{attribute 'GeneratedUsingTerminal: EK1100-0000-0018'}
{attribute addProperty BoxType "EK1100-0000-0018"}
{attribute addProperty Id "Beckhoff_EL2xxxEK1122Beckhoff_EL2xxxEK1122_964E41392A_0001_EL2002_0000_0000EL2002_B02149405A_0002_EL2002_0000_0016EL2002_B02149405A_0003_EL2002_0000_0017EL2002_B02149405A_0004_EL2002_0000_0018EL2002_B02149405A_0005_EL2004_0000_0000EL2004_7B64371E7A_0006_EL2004_0000_0016EL2004_7B64371E7A_0007_EL2004_0000_0017EL2004_7B64371E7A_0008_EL2004_0000_0018EL2004_7B64371E7A_0009_EL2008_0000_0016EL2008_E2806B9511A_0010_EL2008_0000_0017EL2008_E2806B9511A_0011_EL2008_0000_0018EL2008_E2806B9511A_0012_EL2014_0000_0016EL2014_12F3E4E336A_0013_EL2014_0000_0017EL2014_12F3E4E336A_0014_EL2022_0000_0016EL2022_B02149405A_0015_EL2022_0000_0017EL2022_B02149405A_0016_EL2022_0000_0018EL2022_B02149405A_0017_EL2024_0000_0016EL2024_7B64371E7A_0018_EL2024_0000_0017EL2024_7B64371E7A_0019_EL2024_0000_0018EL2024_7B64371E7A_0020_EL2024_0000_0019EL2024_7B64371E7A_0021_EL2024_0010_0016EL2024_7B64371E7A_0022_EL2024_0010_0017EL2024_7B64371E7A_0023_EL2024_0010_0018EL2024_7B64371E7A_0024_EL2032_0000_0000EL2032_4C3AB2A48A_0025_EL2032_0000_0016EL2032_4C3AB2A48A_0026_EL2032_0000_0017EL2032_4C3AB2A48A_0027_EL2032_0000_0018EL2032_4C3AB2A48A_0028_EL2034_0000_0016EL2034_9227BD0712A_0029_EL2034_0000_0017EL2034_9227BD0712A_0030_EL2034_0000_0018EL2034_9227BD0712A_0031_EL2042_0000_0016EL2042_B02149405A_0032_EL2042_0000_0017EL2042_B02149405A_0033_EL2042_0000_0018EL2042_B02149405A_0034_EL2044_0000_0016EL2044_12F3E4E336A_0035_EL2084_0000_0016EL2084_7B64371E7A_0036_EL2084_0000_0017EL2084_7B64371E7A_0037_EL2084_0000_0018EL2084_7B64371E7A_0038_EL2088_0000_0016EL2088_E2806B9511A_0039_EL2088_0000_0017EL2088_E2806B9511A_0040_EL2088_0000_0018EL2088_E2806B9511A_0041_EL2124_0000_0016EL2124_7B64371E7A_0042_EL2124_0000_0017EL2124_7B64371E7A_0043_EL2124_0000_0018EL2124_7B64371E7A_0044_EL2202_0000_0000EL2202_B02149405A_0045_EL2202_0000_0016EL2202_E4D0F2567A_0046_EL2202_0000_0017EL2202_E4D0F2567A_0047_EL2202_0000_0018EL2202_E4D0F2567A_0048_EL2202_0000_0019EL2202_E4D0F2567A_0049_EL2202_0100_0016EL2202_FB12F0C615A_0050_EL2202_0100_0017EL2202_FB12F0C615A_0051_EL2202_0100_0018EL2202_FB12F0C615A_0052_EL2202_0100_0019EL2202_FB12F0C615A_0053_EL2212_0000_0018EL2212_25BC0E0A32A_0054_EL2212_0000_0019EL2212_25BC0E0A32A_0055_EL2212_0000_0020EL2212_C6DE676634A_0056_EL2212_0000_0021EL2212_C6DE676634A_0057_EL2212_0000_0022EL2212_C6DE676634A_0058_EL2212_0000_0023EL2212_C6DE676634A_0059_EL2252_0000_0000EL2252_FF939DB018A_0060_EL2252_0000_0016EL2252_BD1134C622A_0061_EL2252_0000_0017EL2252_F49A8E9224A_0062_EL2252_0000_0018EL2252_F49A8E9224A_0063_EL2252_0000_0019EL2252_F49A8E9224A_0064_EL2252_0000_0020EL2252_F49A8E9224A_0065_EL2258_0000_0016EL2258_1A7A2033508A_0066_EL2258_0000_0017EL2258_41B36B91516A_0067_EL2262_0000_0000EL2262_4683CFC914A_0068_EL2262_0000_0001EL2262_79C970B117A_0069_EL2262_0000_0002EL2262_147DB6E135A_0070_EL2262_0000_0003EL2262_147DB6E135A_0071_EL2262_0000_0004EL2262_9619875D40A_0072_EL2602_0000_0016EL2602_B02149405A_0073_EL2602_0000_0017EL2602_B02149405A_0074_EL2602_0000_0018EL2602_B02149405A_0075_EL2602_0010_0016EL2602_47E63F277A_0076_EL2612_0000_0016EL2612_B02149405A_0077_EL2612_0000_0017EL2612_B02149405A_0078_EL2612_0000_0018EL2612_B02149405A_0079_EL2622_0000_0016EL2622_B02149405A_0080_EL2622_0000_0017EL2622_B02149405A_0081_EL2622_0000_0018EL2622_B02149405A_0082_EL2622_0010_0016EL2622_47E63F277A_0083_EL2624_0000_0016EL2624_7B64371E7A_0084_EL2624_0000_0017EL2624_7B64371E7A_0085_EL2624_0000_0018EL2624_7B64371E7A_0086_EL2634_0000_0016EL2634_7B64371E7A_0087_EL2634_0000_0017EL2634_7B64371E7A_0088_EL2642_0000_0016EL2642_C5F9ACE731A_0089_EL2652_0000_0016EL2652_B02149405A_0090_EL2652_0000_0017EL2652_B02149405A_0091_EL2652_0000_0018EL2652_B02149405A_0092_EL2712_0000_0016EL2712_B02149405A_0093_EL2712_0000_0017EL2712_B02149405A_0094_EL2722_0000_0016EL2722_B02149405A_0095_EL2722_0010_0016EL2722_B02149405A_0096_EL2732_0000_0016EL2732_B02149405A_0097_EL2784_0000_0016EL2784_7B64371E7A_0098_EL2788_0000_0016EL2788_E2806B9511A_0099_EL2794_0000_0016EL2794_7B64371E7A_0100_EL2798_0000_0016EL2798_E2806B9511A_0101_EL2798_0000_0017EL2798_E2806B9511A_0102_EL2798_0000_0018EL2798_E2806B9511A_0103_EL2808_0000_0016EL2808_E2806B9511A_0104_EL2808_0000_0017EL2808_E2806B9511A_0105_EL2808_0000_0018EL2808_E2806B9511A_0106_EL2809_0000_0016EL2809_2B6483BD19A_0107_EL2809_0000_0017EL2809_2B6483BD19A_0108_EL2809_0000_0018EL2809_2B6483BD19A_0109_EL2819_0000_0016EL2819_3C4AB9A796A_0110_EL2819_0000_0017EL2819_3C4AB9A796A_0111_EL2819_0000_0018EL2819_3C4AB9A796A_0112_EL2828_0000_0016EL2828_E2806B9511A_0113_EL2828_0000_0017EL2828_E2806B9511A_0114_EL2872_0000_0016EL2872_2B6483BD19A_0115_EL2872_0000_0017EL2872_2B6483BD19A_0116_EL2872_0000_0018EL2872_2B6483BD19A_0117_EL2872_0000_0019EL2872_2B6483BD19A_0118_EL2872_0010_0016EL2872_2B6483BD19A_0119_EL2872_0010_0017EL2872_2B6483BD19A_0120_EL2872_0010_0018EL2872_2B6483BD19A_0121_EL2872_0010_0019EL2872_2B6483BD19A_0122_EL2878_0005_0016EL2878_76DE585D13A_0123_EL2889_0000_0016EL2889_2B6483BD19A_0124_EL2889_0000_0017EL2889_2B6483BD19A_0125_EL2889_0000_0018EL2889_2B6483BD19A_0126_ELM2642_0000_0016ELM2642_AD2D58FD31A_0127_ELM2644_0000_0016ELM2644_9E566A2A39A_0128_ELM2742_0000_0016ELM2742_AD2D58FD31A_0129_ELM2744_0000_0016ELM2744_9E566A2A39"}
{attribute addProperty CRC "4106566090"}
{attribute addProperty Size "2992"}
TYPE Beckhoff_EL2xxx_F4C539CA EXTENDS EK1100_1FC0878B :
STRUCT
	{attribute addProperty Name "Beckhoff EL2xxxEK1122"}
	{attribute addProperty PreviousPort "Beckhoff EL2xxx : B"}
	Beckhoff_EL2xxxEK1122 : Beckhoff_EL2xxxEK1122_964E4139;
	{attribute addProperty Name "A_0001(EL2002-0000-0000)"}
	{attribute addProperty PreviousPort "Beckhoff EL2xxxEK1122 : C"}
	A_0001_EL2002_0000_0000 : EL2002_B0214940;
	{attribute addProperty Name "A_0002(EL2002-0000-0016)"}
	{attribute addProperty PreviousPort "A_0001(EL2002-0000-0000) : B"}
	A_0002_EL2002_0000_0016 : EL2002_B0214940;
	{attribute addProperty Name "A_0003(EL2002-0000-0017)"}
	{attribute addProperty PreviousPort "A_0002(EL2002-0000-0016) : B"}
	A_0003_EL2002_0000_0017 : EL2002_B0214940;
	{attribute addProperty Name "A_0004(EL2002-0000-0018)"}
	{attribute addProperty PreviousPort "A_0003(EL2002-0000-0017) : B"}
	A_0004_EL2002_0000_0018 : EL2002_B0214940;
	{attribute addProperty Name "A_0005(EL2004-0000-0000)"}
	{attribute addProperty PreviousPort "A_0004(EL2002-0000-0018) : B"}
	A_0005_EL2004_0000_0000 : EL2004_7B64371E;
	{attribute addProperty Name "A_0006(EL2004-0000-0016)"}
	{attribute addProperty PreviousPort "A_0005(EL2004-0000-0000) : B"}
	A_0006_EL2004_0000_0016 : EL2004_7B64371E;
	{attribute addProperty Name "A_0007(EL2004-0000-0017)"}
	{attribute addProperty PreviousPort "A_0006(EL2004-0000-0016) : B"}
	A_0007_EL2004_0000_0017 : EL2004_7B64371E;
	{attribute addProperty Name "A_0008(EL2004-0000-0018)"}
	{attribute addProperty PreviousPort "A_0007(EL2004-0000-0017) : B"}
	A_0008_EL2004_0000_0018 : EL2004_7B64371E;
	{attribute addProperty Name "A_0009(EL2008-0000-0016)"}
	{attribute addProperty PreviousPort "A_0008(EL2004-0000-0018) : B"}
	A_0009_EL2008_0000_0016 : EL2008_E2806B95;
	{attribute addProperty Name "A_0010(EL2008-0000-0017)"}
	{attribute addProperty PreviousPort "A_0009(EL2008-0000-0016) : B"}
	A_0010_EL2008_0000_0017 : EL2008_E2806B95;
	{attribute addProperty Name "A_0011(EL2008-0000-0018)"}
	{attribute addProperty PreviousPort "A_0010(EL2008-0000-0017) : B"}
	A_0011_EL2008_0000_0018 : EL2008_E2806B95;
	{attribute addProperty Name "A_0012(EL2014-0000-0016)"}
	{attribute addProperty PreviousPort "A_0011(EL2008-0000-0018) : B"}
	A_0012_EL2014_0000_0016 : EL2014_12F3E4E3;
	{attribute addProperty Name "A_0013(EL2014-0000-0017)"}
	{attribute addProperty PreviousPort "A_0012(EL2014-0000-0016) : B"}
	A_0013_EL2014_0000_0017 : EL2014_12F3E4E3;
	{attribute addProperty Name "A_0014(EL2022-0000-0016)"}
	{attribute addProperty PreviousPort "A_0013(EL2014-0000-0017) : B"}
	A_0014_EL2022_0000_0016 : EL2022_B0214940;
	{attribute addProperty Name "A_0015(EL2022-0000-0017)"}
	{attribute addProperty PreviousPort "A_0014(EL2022-0000-0016) : B"}
	A_0015_EL2022_0000_0017 : EL2022_B0214940;
	{attribute addProperty Name "A_0016(EL2022-0000-0018)"}
	{attribute addProperty PreviousPort "A_0015(EL2022-0000-0017) : B"}
	A_0016_EL2022_0000_0018 : EL2022_B0214940;
	{attribute addProperty Name "A_0017(EL2024-0000-0016)"}
	{attribute addProperty PreviousPort "A_0016(EL2022-0000-0018) : B"}
	A_0017_EL2024_0000_0016 : EL2024_7B64371E;
	{attribute addProperty Name "A_0018(EL2024-0000-0017)"}
	{attribute addProperty PreviousPort "A_0017(EL2024-0000-0016) : B"}
	A_0018_EL2024_0000_0017 : EL2024_7B64371E;
	{attribute addProperty Name "A_0019(EL2024-0000-0018)"}
	{attribute addProperty PreviousPort "A_0018(EL2024-0000-0017) : B"}
	A_0019_EL2024_0000_0018 : EL2024_7B64371E;
	{attribute addProperty Name "A_0020(EL2024-0000-0019)"}
	{attribute addProperty PreviousPort "A_0019(EL2024-0000-0018) : B"}
	A_0020_EL2024_0000_0019 : EL2024_7B64371E;
	{attribute addProperty Name "A_0021(EL2024-0010-0016)"}
	{attribute addProperty PreviousPort "A_0020(EL2024-0000-0019) : B"}
	A_0021_EL2024_0010_0016 : EL2024_7B64371E;
	{attribute addProperty Name "A_0022(EL2024-0010-0017)"}
	{attribute addProperty PreviousPort "A_0021(EL2024-0010-0016) : B"}
	A_0022_EL2024_0010_0017 : EL2024_7B64371E;
	{attribute addProperty Name "A_0023(EL2024-0010-0018)"}
	{attribute addProperty PreviousPort "A_0022(EL2024-0010-0017) : B"}
	A_0023_EL2024_0010_0018 : EL2024_7B64371E;
	{attribute addProperty Name "A_0024(EL2032-0000-0000)"}
	{attribute addProperty PreviousPort "A_0023(EL2024-0010-0018) : B"}
	A_0024_EL2032_0000_0000 : EL2032_4C3AB2A4;
	{attribute addProperty Name "A_0025(EL2032-0000-0016)"}
	{attribute addProperty PreviousPort "A_0024(EL2032-0000-0000) : B"}
	A_0025_EL2032_0000_0016 : EL2032_4C3AB2A4;
	{attribute addProperty Name "A_0026(EL2032-0000-0017)"}
	{attribute addProperty PreviousPort "A_0025(EL2032-0000-0016) : B"}
	A_0026_EL2032_0000_0017 : EL2032_4C3AB2A4;
	{attribute addProperty Name "A_0027(EL2032-0000-0018)"}
	{attribute addProperty PreviousPort "A_0026(EL2032-0000-0017) : B"}
	A_0027_EL2032_0000_0018 : EL2032_4C3AB2A4;
	{attribute addProperty Name "A_0028(EL2034-0000-0016)"}
	{attribute addProperty PreviousPort "A_0027(EL2032-0000-0018) : B"}
	A_0028_EL2034_0000_0016 : EL2034_9227BD07;
	{attribute addProperty Name "A_0029(EL2034-0000-0017)"}
	{attribute addProperty PreviousPort "A_0028(EL2034-0000-0016) : B"}
	A_0029_EL2034_0000_0017 : EL2034_9227BD07;
	{attribute addProperty Name "A_0030(EL2034-0000-0018)"}
	{attribute addProperty PreviousPort "A_0029(EL2034-0000-0017) : B"}
	A_0030_EL2034_0000_0018 : EL2034_9227BD07;
	{attribute addProperty Name "A_0031(EL2042-0000-0016)"}
	{attribute addProperty PreviousPort "A_0030(EL2034-0000-0018) : B"}
	A_0031_EL2042_0000_0016 : EL2042_B0214940;
	{attribute addProperty Name "A_0032(EL2042-0000-0017)"}
	{attribute addProperty PreviousPort "A_0031(EL2042-0000-0016) : B"}
	A_0032_EL2042_0000_0017 : EL2042_B0214940;
	{attribute addProperty Name "A_0033(EL2042-0000-0018)"}
	{attribute addProperty PreviousPort "A_0032(EL2042-0000-0017) : B"}
	A_0033_EL2042_0000_0018 : EL2042_B0214940;
	{attribute addProperty Name "A_0034(EL2044-0000-0016)"}
	{attribute addProperty PreviousPort "A_0033(EL2042-0000-0018) : B"}
	A_0034_EL2044_0000_0016 : EL2044_12F3E4E3;
	{attribute addProperty Name "A_0035(EL2084-0000-0016)"}
	{attribute addProperty PreviousPort "A_0034(EL2044-0000-0016) : B"}
	A_0035_EL2084_0000_0016 : EL2084_7B64371E;
	{attribute addProperty Name "A_0036(EL2084-0000-0017)"}
	{attribute addProperty PreviousPort "A_0035(EL2084-0000-0016) : B"}
	A_0036_EL2084_0000_0017 : EL2084_7B64371E;
	{attribute addProperty Name "A_0037(EL2084-0000-0018)"}
	{attribute addProperty PreviousPort "A_0036(EL2084-0000-0017) : B"}
	A_0037_EL2084_0000_0018 : EL2084_7B64371E;
	{attribute addProperty Name "A_0038(EL2088-0000-0016)"}
	{attribute addProperty PreviousPort "A_0037(EL2084-0000-0018) : B"}
	A_0038_EL2088_0000_0016 : EL2088_E2806B95;
	{attribute addProperty Name "A_0039(EL2088-0000-0017)"}
	{attribute addProperty PreviousPort "A_0038(EL2088-0000-0016) : B"}
	A_0039_EL2088_0000_0017 : EL2088_E2806B95;
	{attribute addProperty Name "A_0040(EL2088-0000-0018)"}
	{attribute addProperty PreviousPort "A_0039(EL2088-0000-0017) : B"}
	A_0040_EL2088_0000_0018 : EL2088_E2806B95;
	{attribute addProperty Name "A_0041(EL2124-0000-0016)"}
	{attribute addProperty PreviousPort "A_0040(EL2088-0000-0018) : B"}
	A_0041_EL2124_0000_0016 : EL2124_7B64371E;
	{attribute addProperty Name "A_0042(EL2124-0000-0017)"}
	{attribute addProperty PreviousPort "A_0041(EL2124-0000-0016) : B"}
	A_0042_EL2124_0000_0017 : EL2124_7B64371E;
	{attribute addProperty Name "A_0043(EL2124-0000-0018)"}
	{attribute addProperty PreviousPort "A_0042(EL2124-0000-0017) : B"}
	A_0043_EL2124_0000_0018 : EL2124_7B64371E;
	{attribute addProperty Name "A_0044(EL2202-0000-0000)"}
	{attribute addProperty PreviousPort "A_0043(EL2124-0000-0018) : B"}
	A_0044_EL2202_0000_0000 : EL2202_B0214940;
	{attribute addProperty Name "A_0045(EL2202-0000-0016)"}
	{attribute addProperty PreviousPort "A_0044(EL2202-0000-0000) : B"}
	A_0045_EL2202_0000_0016 : EL2202_E4D0F256;
	{attribute addProperty Name "A_0046(EL2202-0000-0017)"}
	{attribute addProperty PreviousPort "A_0045(EL2202-0000-0016) : B"}
	A_0046_EL2202_0000_0017 : EL2202_E4D0F256;
	{attribute addProperty Name "A_0047(EL2202-0000-0018)"}
	{attribute addProperty PreviousPort "A_0046(EL2202-0000-0017) : B"}
	A_0047_EL2202_0000_0018 : EL2202_E4D0F256;
	{attribute addProperty Name "A_0048(EL2202-0000-0019)"}
	{attribute addProperty PreviousPort "A_0047(EL2202-0000-0018) : B"}
	A_0048_EL2202_0000_0019 : EL2202_E4D0F256;
	{attribute addProperty Name "A_0049(EL2202-0100-0016)"}
	{attribute addProperty PreviousPort "A_0048(EL2202-0000-0019) : B"}
	A_0049_EL2202_0100_0016 : EL2202_FB12F0C6;
	{attribute addProperty Name "A_0050(EL2202-0100-0017)"}
	{attribute addProperty PreviousPort "A_0049(EL2202-0100-0016) : B"}
	A_0050_EL2202_0100_0017 : EL2202_FB12F0C6;
	{attribute addProperty Name "A_0051(EL2202-0100-0018)"}
	{attribute addProperty PreviousPort "A_0050(EL2202-0100-0017) : B"}
	A_0051_EL2202_0100_0018 : EL2202_FB12F0C6;
	{attribute addProperty Name "A_0052(EL2202-0100-0019)"}
	{attribute addProperty PreviousPort "A_0051(EL2202-0100-0018) : B"}
	A_0052_EL2202_0100_0019 : EL2202_FB12F0C6;
	{attribute addProperty Name "A_0053(EL2212-0000-0018)"}
	{attribute addProperty PreviousPort "A_0052(EL2202-0100-0019) : B"}
	A_0053_EL2212_0000_0018 : EL2212_25BC0E0A;
	{attribute addProperty Name "A_0054(EL2212-0000-0019)"}
	{attribute addProperty PreviousPort "A_0053(EL2212-0000-0018) : B"}
	A_0054_EL2212_0000_0019 : EL2212_25BC0E0A;
	{attribute addProperty Name "A_0055(EL2212-0000-0020)"}
	{attribute addProperty PreviousPort "A_0054(EL2212-0000-0019) : B"}
	A_0055_EL2212_0000_0020 : EL2212_C6DE6766;
	{attribute addProperty Name "A_0056(EL2212-0000-0021)"}
	{attribute addProperty PreviousPort "A_0055(EL2212-0000-0020) : B"}
	A_0056_EL2212_0000_0021 : EL2212_C6DE6766;
	{attribute addProperty Name "A_0057(EL2212-0000-0022)"}
	{attribute addProperty PreviousPort "A_0056(EL2212-0000-0021) : B"}
	A_0057_EL2212_0000_0022 : EL2212_C6DE6766;
	{attribute addProperty Name "A_0058(EL2212-0000-0023)"}
	{attribute addProperty PreviousPort "A_0057(EL2212-0000-0022) : B"}
	A_0058_EL2212_0000_0023 : EL2212_C6DE6766;
	{attribute addProperty Name "A_0059(EL2252-0000-0000)"}
	{attribute addProperty PreviousPort "A_0058(EL2212-0000-0023) : B"}
	A_0059_EL2252_0000_0000 : EL2252_FF939DB0;
	{attribute addProperty Name "A_0060(EL2252-0000-0016)"}
	{attribute addProperty PreviousPort "A_0059(EL2252-0000-0000) : B"}
	A_0060_EL2252_0000_0016 : EL2252_BD1134C6;
	{attribute addProperty Name "A_0061(EL2252-0000-0017)"}
	{attribute addProperty PreviousPort "A_0060(EL2252-0000-0016) : B"}
	A_0061_EL2252_0000_0017 : EL2252_F49A8E92;
	{attribute addProperty Name "A_0062(EL2252-0000-0018)"}
	{attribute addProperty PreviousPort "A_0061(EL2252-0000-0017) : B"}
	A_0062_EL2252_0000_0018 : EL2252_F49A8E92;
	{attribute addProperty Name "A_0063(EL2252-0000-0019)"}
	{attribute addProperty PreviousPort "A_0062(EL2252-0000-0018) : B"}
	A_0063_EL2252_0000_0019 : EL2252_F49A8E92;
	{attribute addProperty Name "A_0064(EL2252-0000-0020)"}
	{attribute addProperty PreviousPort "A_0063(EL2252-0000-0019) : B"}
	A_0064_EL2252_0000_0020 : EL2252_F49A8E92;
	{attribute addProperty Name "A_0065(EL2258-0000-0016)"}
	{attribute addProperty PreviousPort "A_0064(EL2252-0000-0020) : B"}
	A_0065_EL2258_0000_0016 : EL2258_1A7A2033;
	{attribute addProperty Name "A_0066(EL2258-0000-0017)"}
	{attribute addProperty PreviousPort "A_0065(EL2258-0000-0016) : B"}
	A_0066_EL2258_0000_0017 : EL2258_41B36B91;
	{attribute addProperty Name "A_0067(EL2262-0000-0000)"}
	{attribute addProperty PreviousPort "A_0066(EL2258-0000-0017) : B"}
	A_0067_EL2262_0000_0000 : EL2262_4683CFC9;
	{attribute addProperty Name "A_0068(EL2262-0000-0001)"}
	{attribute addProperty PreviousPort "A_0067(EL2262-0000-0000) : B"}
	A_0068_EL2262_0000_0001 : EL2262_79C970B1;
	{attribute addProperty Name "A_0069(EL2262-0000-0002)"}
	{attribute addProperty PreviousPort "A_0068(EL2262-0000-0001) : B"}
	A_0069_EL2262_0000_0002 : EL2262_147DB6E1;
	{attribute addProperty Name "A_0070(EL2262-0000-0003)"}
	{attribute addProperty PreviousPort "A_0069(EL2262-0000-0002) : B"}
	A_0070_EL2262_0000_0003 : EL2262_147DB6E1;
	{attribute addProperty Name "A_0071(EL2262-0000-0004)"}
	{attribute addProperty PreviousPort "A_0070(EL2262-0000-0003) : B"}
	A_0071_EL2262_0000_0004 : EL2262_9619875D;
	{attribute addProperty Name "A_0072(EL2602-0000-0016)"}
	{attribute addProperty PreviousPort "A_0071(EL2262-0000-0004) : B"}
	A_0072_EL2602_0000_0016 : EL2602_B0214940;
	{attribute addProperty Name "A_0073(EL2602-0000-0017)"}
	{attribute addProperty PreviousPort "A_0072(EL2602-0000-0016) : B"}
	A_0073_EL2602_0000_0017 : EL2602_B0214940;
	{attribute addProperty Name "A_0074(EL2602-0000-0018)"}
	{attribute addProperty PreviousPort "A_0073(EL2602-0000-0017) : B"}
	A_0074_EL2602_0000_0018 : EL2602_B0214940;
	{attribute addProperty Name "A_0075(EL2602-0010-0016)"}
	{attribute addProperty PreviousPort "A_0074(EL2602-0000-0018) : B"}
	A_0075_EL2602_0010_0016 : EL2602_47E63F27;
	{attribute addProperty Name "A_0076(EL2612-0000-0016)"}
	{attribute addProperty PreviousPort "A_0075(EL2602-0010-0016) : B"}
	A_0076_EL2612_0000_0016 : EL2612_B0214940;
	{attribute addProperty Name "A_0077(EL2612-0000-0017)"}
	{attribute addProperty PreviousPort "A_0076(EL2612-0000-0016) : B"}
	A_0077_EL2612_0000_0017 : EL2612_B0214940;
	{attribute addProperty Name "A_0078(EL2612-0000-0018)"}
	{attribute addProperty PreviousPort "A_0077(EL2612-0000-0017) : B"}
	A_0078_EL2612_0000_0018 : EL2612_B0214940;
	{attribute addProperty Name "A_0079(EL2622-0000-0016)"}
	{attribute addProperty PreviousPort "A_0078(EL2612-0000-0018) : B"}
	A_0079_EL2622_0000_0016 : EL2622_B0214940;
	{attribute addProperty Name "A_0080(EL2622-0000-0017)"}
	{attribute addProperty PreviousPort "A_0079(EL2622-0000-0016) : B"}
	A_0080_EL2622_0000_0017 : EL2622_B0214940;
	{attribute addProperty Name "A_0081(EL2622-0000-0018)"}
	{attribute addProperty PreviousPort "A_0080(EL2622-0000-0017) : B"}
	A_0081_EL2622_0000_0018 : EL2622_B0214940;
	{attribute addProperty Name "A_0082(EL2622-0010-0016)"}
	{attribute addProperty PreviousPort "A_0081(EL2622-0000-0018) : B"}
	A_0082_EL2622_0010_0016 : EL2622_47E63F27;
	{attribute addProperty Name "A_0083(EL2624-0000-0016)"}
	{attribute addProperty PreviousPort "A_0082(EL2622-0010-0016) : B"}
	A_0083_EL2624_0000_0016 : EL2624_7B64371E;
	{attribute addProperty Name "A_0084(EL2624-0000-0017)"}
	{attribute addProperty PreviousPort "A_0083(EL2624-0000-0016) : B"}
	A_0084_EL2624_0000_0017 : EL2624_7B64371E;
	{attribute addProperty Name "A_0085(EL2624-0000-0018)"}
	{attribute addProperty PreviousPort "A_0084(EL2624-0000-0017) : B"}
	A_0085_EL2624_0000_0018 : EL2624_7B64371E;
	{attribute addProperty Name "A_0086(EL2634-0000-0016)"}
	{attribute addProperty PreviousPort "A_0085(EL2624-0000-0018) : B"}
	A_0086_EL2634_0000_0016 : EL2634_7B64371E;
	{attribute addProperty Name "A_0087(EL2634-0000-0017)"}
	{attribute addProperty PreviousPort "A_0086(EL2634-0000-0016) : B"}
	A_0087_EL2634_0000_0017 : EL2634_7B64371E;
	{attribute addProperty Name "A_0088(EL2642-0000-0016)"}
	{attribute addProperty PreviousPort "A_0087(EL2634-0000-0017) : B"}
	A_0088_EL2642_0000_0016 : EL2642_C5F9ACE7;
	{attribute addProperty Name "A_0089(EL2652-0000-0016)"}
	{attribute addProperty PreviousPort "A_0088(EL2642-0000-0016) : B"}
	A_0089_EL2652_0000_0016 : EL2652_B0214940;
	{attribute addProperty Name "A_0090(EL2652-0000-0017)"}
	{attribute addProperty PreviousPort "A_0089(EL2652-0000-0016) : B"}
	A_0090_EL2652_0000_0017 : EL2652_B0214940;
	{attribute addProperty Name "A_0091(EL2652-0000-0018)"}
	{attribute addProperty PreviousPort "A_0090(EL2652-0000-0017) : B"}
	A_0091_EL2652_0000_0018 : EL2652_B0214940;
	{attribute addProperty Name "A_0092(EL2712-0000-0016)"}
	{attribute addProperty PreviousPort "A_0091(EL2652-0000-0018) : B"}
	A_0092_EL2712_0000_0016 : EL2712_B0214940;
	{attribute addProperty Name "A_0093(EL2712-0000-0017)"}
	{attribute addProperty PreviousPort "A_0092(EL2712-0000-0016) : B"}
	A_0093_EL2712_0000_0017 : EL2712_B0214940;
	{attribute addProperty Name "A_0094(EL2722-0000-0016)"}
	{attribute addProperty PreviousPort "A_0093(EL2712-0000-0017) : B"}
	A_0094_EL2722_0000_0016 : EL2722_B0214940;
	{attribute addProperty Name "A_0095(EL2722-0010-0016)"}
	{attribute addProperty PreviousPort "A_0094(EL2722-0000-0016) : B"}
	A_0095_EL2722_0010_0016 : EL2722_B0214940;
	{attribute addProperty Name "A_0096(EL2732-0000-0016)"}
	{attribute addProperty PreviousPort "A_0095(EL2722-0010-0016) : B"}
	A_0096_EL2732_0000_0016 : EL2732_B0214940;
	{attribute addProperty Name "A_0097(EL2784-0000-0016)"}
	{attribute addProperty PreviousPort "A_0096(EL2732-0000-0016) : B"}
	A_0097_EL2784_0000_0016 : EL2784_7B64371E;
	{attribute addProperty Name "A_0098(EL2788-0000-0016)"}
	{attribute addProperty PreviousPort "A_0097(EL2784-0000-0016) : B"}
	A_0098_EL2788_0000_0016 : EL2788_E2806B95;
	{attribute addProperty Name "A_0099(EL2794-0000-0016)"}
	{attribute addProperty PreviousPort "A_0098(EL2788-0000-0016) : B"}
	A_0099_EL2794_0000_0016 : EL2794_7B64371E;
	{attribute addProperty Name "A_0100(EL2798-0000-0016)"}
	{attribute addProperty PreviousPort "A_0099(EL2794-0000-0016) : B"}
	A_0100_EL2798_0000_0016 : EL2798_E2806B95;
	{attribute addProperty Name "A_0101(EL2798-0000-0017)"}
	{attribute addProperty PreviousPort "A_0100(EL2798-0000-0016) : B"}
	A_0101_EL2798_0000_0017 : EL2798_E2806B95;
	{attribute addProperty Name "A_0102(EL2798-0000-0018)"}
	{attribute addProperty PreviousPort "A_0101(EL2798-0000-0017) : B"}
	A_0102_EL2798_0000_0018 : EL2798_E2806B95;
	{attribute addProperty Name "A_0103(EL2808-0000-0016)"}
	{attribute addProperty PreviousPort "A_0102(EL2798-0000-0018) : B"}
	A_0103_EL2808_0000_0016 : EL2808_E2806B95;
	{attribute addProperty Name "A_0104(EL2808-0000-0017)"}
	{attribute addProperty PreviousPort "A_0103(EL2808-0000-0016) : B"}
	A_0104_EL2808_0000_0017 : EL2808_E2806B95;
	{attribute addProperty Name "A_0105(EL2808-0000-0018)"}
	{attribute addProperty PreviousPort "A_0104(EL2808-0000-0017) : B"}
	A_0105_EL2808_0000_0018 : EL2808_E2806B95;
	{attribute addProperty Name "A_0106(EL2809-0000-0016)"}
	{attribute addProperty PreviousPort "A_0105(EL2808-0000-0018) : B"}
	A_0106_EL2809_0000_0016 : EL2809_2B6483BD;
	{attribute addProperty Name "A_0107(EL2809-0000-0017)"}
	{attribute addProperty PreviousPort "A_0106(EL2809-0000-0016) : B"}
	A_0107_EL2809_0000_0017 : EL2809_2B6483BD;
	{attribute addProperty Name "A_0108(EL2809-0000-0018)"}
	{attribute addProperty PreviousPort "A_0107(EL2809-0000-0017) : B"}
	A_0108_EL2809_0000_0018 : EL2809_2B6483BD;
	{attribute addProperty Name "A_0109(EL2819-0000-0016)"}
	{attribute addProperty PreviousPort "A_0108(EL2809-0000-0018) : B"}
	A_0109_EL2819_0000_0016 : EL2819_3C4AB9A7;
	{attribute addProperty Name "A_0110(EL2819-0000-0017)"}
	{attribute addProperty PreviousPort "A_0109(EL2819-0000-0016) : B"}
	A_0110_EL2819_0000_0017 : EL2819_3C4AB9A7;
	{attribute addProperty Name "A_0111(EL2819-0000-0018)"}
	{attribute addProperty PreviousPort "A_0110(EL2819-0000-0017) : B"}
	A_0111_EL2819_0000_0018 : EL2819_3C4AB9A7;
	{attribute addProperty Name "A_0112(EL2828-0000-0016)"}
	{attribute addProperty PreviousPort "A_0111(EL2819-0000-0018) : B"}
	A_0112_EL2828_0000_0016 : EL2828_E2806B95;
	{attribute addProperty Name "A_0113(EL2828-0000-0017)"}
	{attribute addProperty PreviousPort "A_0112(EL2828-0000-0016) : B"}
	A_0113_EL2828_0000_0017 : EL2828_E2806B95;
	{attribute addProperty Name "A_0114(EL2872-0000-0016)"}
	{attribute addProperty PreviousPort "A_0113(EL2828-0000-0017) : B"}
	A_0114_EL2872_0000_0016 : EL2872_2B6483BD;
	{attribute addProperty Name "A_0115(EL2872-0000-0017)"}
	{attribute addProperty PreviousPort "A_0114(EL2872-0000-0016) : B"}
	A_0115_EL2872_0000_0017 : EL2872_2B6483BD;
	{attribute addProperty Name "A_0116(EL2872-0000-0018)"}
	{attribute addProperty PreviousPort "A_0115(EL2872-0000-0017) : B"}
	A_0116_EL2872_0000_0018 : EL2872_2B6483BD;
	{attribute addProperty Name "A_0117(EL2872-0000-0019)"}
	{attribute addProperty PreviousPort "A_0116(EL2872-0000-0018) : B"}
	A_0117_EL2872_0000_0019 : EL2872_2B6483BD;
	{attribute addProperty Name "A_0118(EL2872-0010-0016)"}
	{attribute addProperty PreviousPort "A_0117(EL2872-0000-0019) : B"}
	A_0118_EL2872_0010_0016 : EL2872_2B6483BD;
	{attribute addProperty Name "A_0119(EL2872-0010-0017)"}
	{attribute addProperty PreviousPort "A_0118(EL2872-0010-0016) : B"}
	A_0119_EL2872_0010_0017 : EL2872_2B6483BD;
	{attribute addProperty Name "A_0120(EL2872-0010-0018)"}
	{attribute addProperty PreviousPort "A_0119(EL2872-0010-0017) : B"}
	A_0120_EL2872_0010_0018 : EL2872_2B6483BD;
	{attribute addProperty Name "A_0121(EL2872-0010-0019)"}
	{attribute addProperty PreviousPort "A_0120(EL2872-0010-0018) : B"}
	A_0121_EL2872_0010_0019 : EL2872_2B6483BD;
	{attribute addProperty Name "A_0122(EL2878-0005-0016)"}
	{attribute addProperty PreviousPort "A_0121(EL2872-0010-0019) : B"}
	A_0122_EL2878_0005_0016 : EL2878_76DE585D;
	{attribute addProperty Name "A_0123(EL2889-0000-0016)"}
	{attribute addProperty PreviousPort "A_0122(EL2878-0005-0016) : B"}
	A_0123_EL2889_0000_0016 : EL2889_2B6483BD;
	{attribute addProperty Name "A_0124(EL2889-0000-0017)"}
	{attribute addProperty PreviousPort "A_0123(EL2889-0000-0016) : B"}
	A_0124_EL2889_0000_0017 : EL2889_2B6483BD;
	{attribute addProperty Name "A_0125(EL2889-0000-0018)"}
	{attribute addProperty PreviousPort "A_0124(EL2889-0000-0017) : B"}
	A_0125_EL2889_0000_0018 : EL2889_2B6483BD;
	{attribute addProperty Name "A_0126(ELM2642-0000-0016)"}
	{attribute addProperty PreviousPort "A_0125(EL2889-0000-0018) : B"}
	A_0126_ELM2642_0000_0016 : ELM2642_AD2D58FD;
	{attribute addProperty Name "A_0127(ELM2644-0000-0016)"}
	{attribute addProperty PreviousPort "A_0126(ELM2642-0000-0016) : B"}
	A_0127_ELM2644_0000_0016 : ELM2644_9E566A2A;
	{attribute addProperty Name "A_0128(ELM2742-0000-0016)"}
	{attribute addProperty PreviousPort "A_0127(ELM2644-0000-0016) : B"}
	A_0128_ELM2742_0000_0016 : ELM2742_AD2D58FD;
	{attribute addProperty Name "A_0129(ELM2744-0000-0016)"}
	{attribute addProperty PreviousPort "A_0128(ELM2742-0000-0016) : B"}
	A_0129_ELM2744_0000_0016 : ELM2744_9E566A2A;
END_STRUCT
END_TYPE

(* stored: Version 1.2.0.0, ProductVersion 3.1.4024.9
   DUT Beckhoff_EL2xxx_F4C539CA: Id {40a5cad6-06c0-478c-9478-dfab246f972e} *)
